TYPE ST_DI :
STRUCT
		Value		  AT %I*	: BOOL	;
		Description 			: STRING	;

END_STRUCT
END_TYPE

(* stored: Version 1.1.0.1, ProductVersion 3.1.4022.11
   DUT ST_DI: Id {ee7faff8-d538-4cb9-a9ed-a99e04cbeea3} *)
